% RSLogix 500 project FINAL PROJECT_thisone.RSS, saved by version 8.30.00.16 %
PROJECT "UNTITLED"    % processor: MicroLogix 1000 %

PROGRAM FILES
  LAD 2 "MAIN_PROG"  27 rungs
  LAD 3 "USER_FAULT"  1 rungs
  LAD 4 "HSC_INT"  1 rungs
  LAD 5 "STI_INT"  1 rungs
  LAD 6, 7, 8, 9, 10, 11, 12, 13, 14, 15, 16: only END

DATA FILES
  O0 OUTPUT  1 elements
  I1 INPUT  2 elements
  S2 STATUS  33 elements
  B3 BINARY  32 elements
  T4 TIMER  40 elements
  C5 COUNTER  32 elements
  R6 CONTROL  16 elements
  N7 INTEGER  105 elements

LADDER 2 "MAIN_PROG"
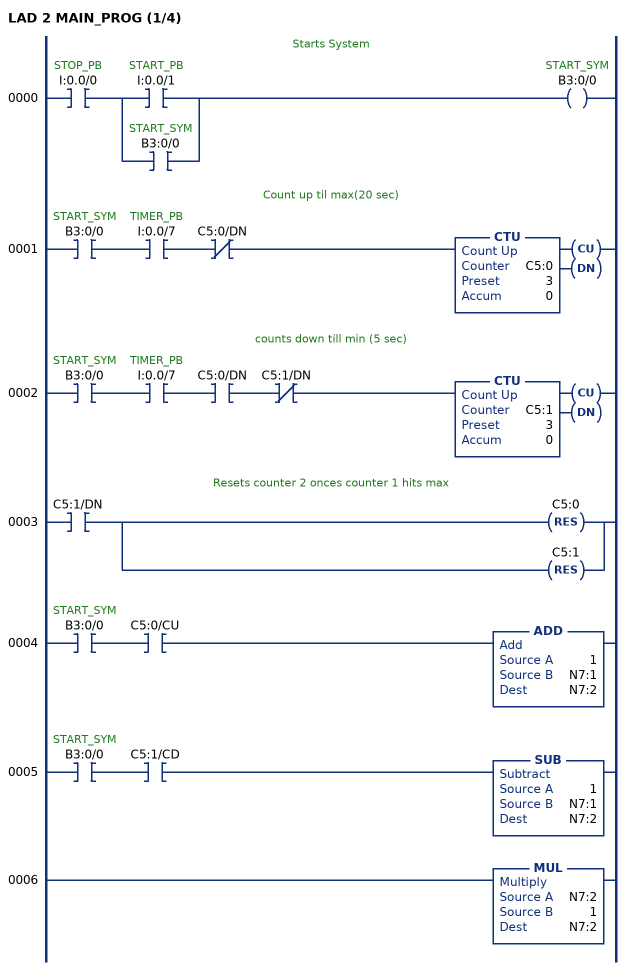
% Rung: 0 %
% Starts System %
SOR XIC I:0.0/0 BST XIC I:0.0/1 NXB XIC B3:0/0 BND OTE B3:0/0 EOR
%   I:0.0/0  STOP_PB %
%   I:0.0/1  START_PB %
%   B3:0/0  START_SYM %
% Rung: 1 %
% Count up til max(20 sec) %
SOR XIC B3:0/0 XIC I:0.0/7 XIO C5:0/DN CTU C5:0 3 0 EOR
%   B3:0/0  START_SYM %
%   I:0.0/7  TIMER_PB %
% Rung: 2 %
% counts down till min (5 sec) %
SOR XIC B3:0/0 XIC I:0.0/7 XIC C5:0/DN XIO C5:1/DN CTU C5:1 3 0 EOR
%   B3:0/0  START_SYM %
%   I:0.0/7  TIMER_PB %
% Rung: 3 %
% Resets counter 2 onces counter 1 hits max %
SOR XIC C5:1/DN BST RES C5:0 NXB RES C5:1 BND EOR
% Rung: 4 %
SOR XIC B3:0/0 XIC C5:0/CU ADD 1 N7:1 N7:2 EOR
%   B3:0/0  START_SYM %
% Rung: 5 %
SOR XIC B3:0/0 XIC C5:1/CD SUB 1 N7:1 N7:2 EOR
%   B3:0/0  START_SYM %
% Rung: 6 %
SOR MUL N7:2 1 N7:2 EOR

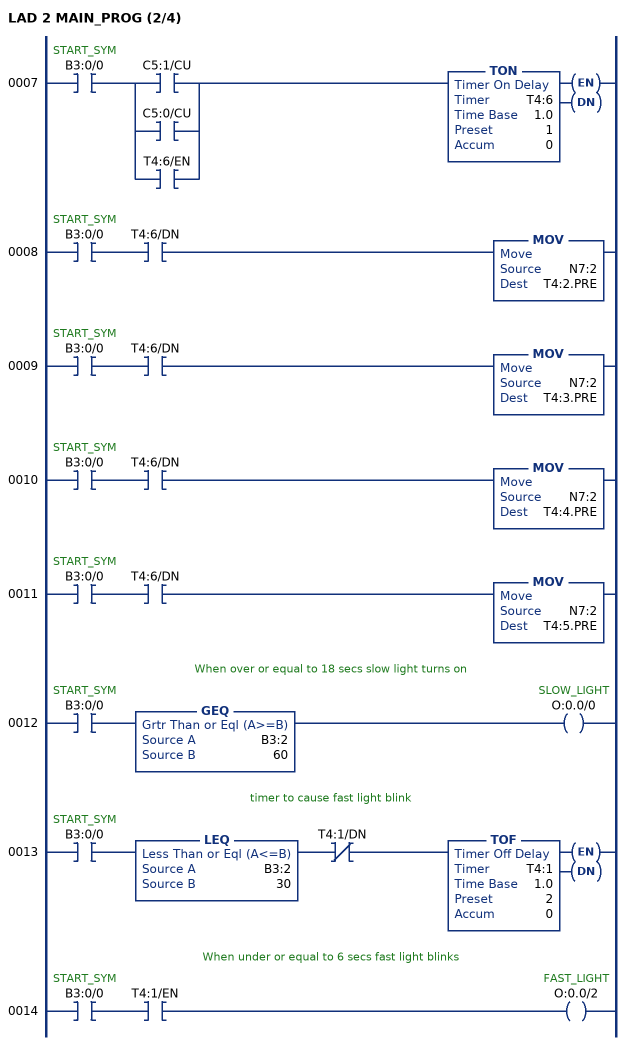
% Rung: 7 %
SOR XIC B3:0/0 BST XIC C5:1/CU NXB XIC C5:0/CU NXB XIC T4:6/EN BND TON T4:6 1.0 1 0 EOR
%   B3:0/0  START_SYM %
% Rung: 8 %
SOR XIC B3:0/0 XIC T4:6/DN MOV N7:2 T4:2.PRE EOR
%   B3:0/0  START_SYM %
% Rung: 9 %
SOR XIC B3:0/0 XIC T4:6/DN MOV N7:2 T4:3.PRE EOR
%   B3:0/0  START_SYM %
% Rung: 10 %
SOR XIC B3:0/0 XIC T4:6/DN MOV N7:2 T4:4.PRE EOR
%   B3:0/0  START_SYM %
% Rung: 11 %
SOR XIC B3:0/0 XIC T4:6/DN MOV N7:2 T4:5.PRE EOR
%   B3:0/0  START_SYM %
% Rung: 12 %
% When over or equal to 18 secs slow light turns on %
SOR XIC B3:0/0 GEQ B3:2 60 OTE O:0.0/0 EOR
%   B3:0/0  START_SYM %
%   O:0.0/0  SLOW_LIGHT %
% Rung: 13 %
% timer to cause fast light blink %
SOR XIC B3:0/0 LEQ B3:2 30 XIO T4:1/DN TOF T4:1 1.0 2 0 EOR
%   B3:0/0  START_SYM %
% Rung: 14 %
% When under or equal to 6 secs fast light blinks %
SOR XIC B3:0/0 XIC T4:1/EN OTE O:0.0/2 EOR
%   B3:0/0  START_SYM %
%   O:0.0/2  FAST_LIGHT %

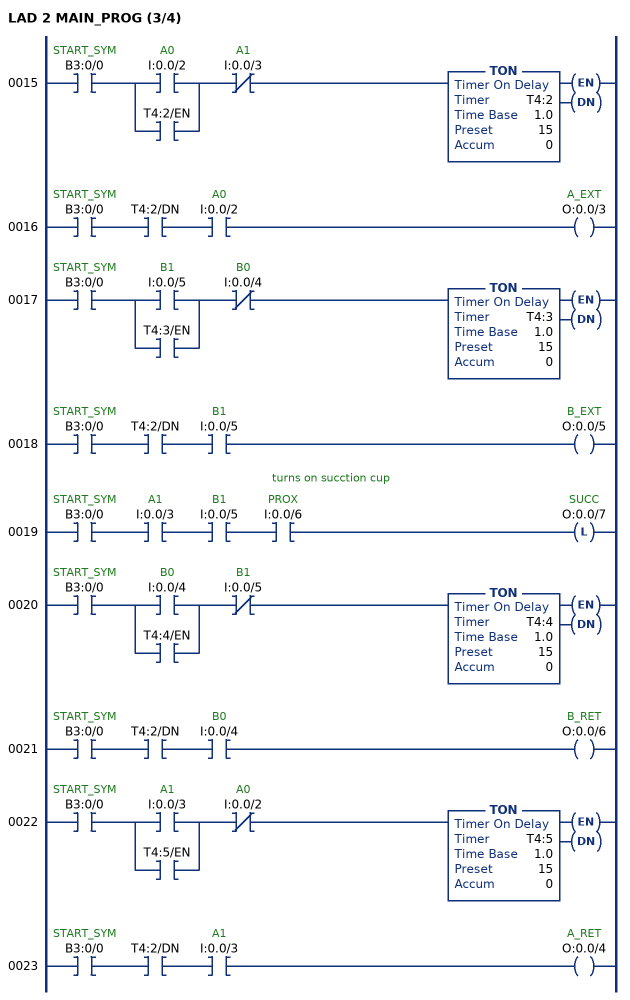
% Rung: 15 %
SOR XIC B3:0/0 BST XIC I:0.0/2 NXB XIC T4:2/EN BND XIO I:0.0/3 TON T4:2 1.0 15 0 EOR
%   B3:0/0  START_SYM %
%   I:0.0/2  A0 %
%   I:0.0/3  A1 %
% Rung: 16 %
SOR XIC B3:0/0 XIC T4:2/DN XIC I:0.0/2 OTE O:0.0/3 EOR
%   B3:0/0  START_SYM %
%   I:0.0/2  A0 %
%   O:0.0/3  A_EXT %
% Rung: 17 %
SOR XIC B3:0/0 BST XIC I:0.0/5 NXB XIC T4:3/EN BND XIO I:0.0/4 TON T4:3 1.0 15 0 EOR
%   B3:0/0  START_SYM %
%   I:0.0/5  B1 %
%   I:0.0/4  B0 %
% Rung: 18 %
SOR XIC B3:0/0 XIC T4:2/DN XIC I:0.0/5 OTE O:0.0/5 EOR
%   B3:0/0  START_SYM %
%   I:0.0/5  B1 %
%   O:0.0/5  B_EXT %
% Rung: 19 %
% turns on sucction cup %
SOR XIC B3:0/0 XIC I:0.0/3 XIC I:0.0/5 XIC I:0.0/6 OTL O:0.0/7 EOR
%   B3:0/0  START_SYM %
%   I:0.0/3  A1 %
%   I:0.0/5  B1 %
%   I:0.0/6  PROX %
%   O:0.0/7  SUCC %
% Rung: 20 %
SOR XIC B3:0/0 BST XIC I:0.0/4 NXB XIC T4:4/EN BND XIO I:0.0/5 TON T4:4 1.0 15 0 EOR
%   B3:0/0  START_SYM %
%   I:0.0/4  B0 %
%   I:0.0/5  B1 %
% Rung: 21 %
SOR XIC B3:0/0 XIC T4:2/DN XIC I:0.0/4 OTE O:0.0/6 EOR
%   B3:0/0  START_SYM %
%   I:0.0/4  B0 %
%   O:0.0/6  B_RET %
% Rung: 22 %
SOR XIC B3:0/0 BST XIC I:0.0/3 NXB XIC T4:5/EN BND XIO I:0.0/2 TON T4:5 1.0 15 0 EOR
%   B3:0/0  START_SYM %
%   I:0.0/3  A1 %
%   I:0.0/2  A0 %
% Rung: 23 %
SOR XIC B3:0/0 XIC T4:2/DN XIC I:0.0/3 OTE O:0.0/4 EOR
%   B3:0/0  START_SYM %
%   I:0.0/3  A1 %
%   O:0.0/4  A_RET %

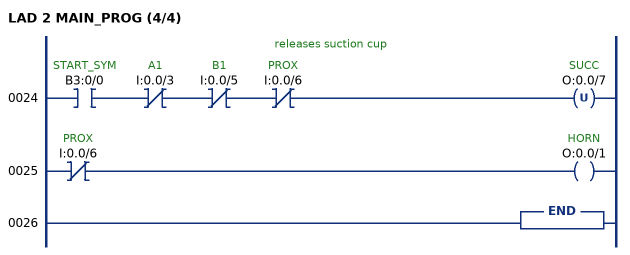
% Rung: 24 %
% releases suction cup %
SOR XIC B3:0/0 XIO I:0.0/3 XIO I:0.0/5 XIO I:0.0/6 OTU O:0.0/7 EOR
%   B3:0/0  START_SYM %
%   I:0.0/3  A1 %
%   I:0.0/5  B1 %
%   I:0.0/6  PROX %
%   O:0.0/7  SUCC %
% Rung: 25 %
SOR XIO I:0.0/6 OTE O:0.0/1 EOR
%   I:0.0/6  PROX %
%   O:0.0/1  HORN %
% Rung: 26 %
SOR END EOR

OTHER DOCUMENTED ADDRESSES
  T0:0  T0

COMMENTS NOT ATTACHED TO A CURRENT RUNG
  C5:0: Resets counter 1 onces counter 2 hits max
  T4:0: Timer Pushbutton with delay
  B3:0/0: Starts System

DATA TABLE (non-zero values as saved)
DATA T4
% .PRE .ACC %
% T4:0 % 1 0
% T4:1 % 2 0
% T4:2 % 15 0
% T4:3 % 15 0
% T4:4 % 15 0
% T4:5 % 15 0
% T4:6 % 1 0
% T4:8 % 1 0
% T4:9 % 1 0
DATA C5
% .PRE .ACC %
% C5:0 % 3 0
% C5:1 % 3 0
